DATA_BLOCK "RSE_DB"
TITLE = Report System Error Diagnostic Block
{ S7_Optimized_Access := 'FALSE' }
AUTHOR : SIMATIC
FAMILY : RSEDIAG
NAME : RSE4
VERSION : 1.0
NON_RETAIN
// This DB contains the generated data from STEP 7 Report System Errors.
"RSE_FB"

BEGIN
   w127Timer_a := BYTE#16#80;
   bAnwenderIO_Flag := BYTE#16#54;
   wRackEntry1 := WORD#16#0368;
   xFrei := TRUE;
   VFTable0_Hiera := BYTE#16#01;
   VFTable0_AsyncFct := BYTE#16#07;
   VFTable0_AsyncDat := BYTE#16#0F;
   VFTable0_SyncFct := BYTE#16#07;
   VFTable0_SyncDat := BYTE#16#0F;
   VFTable0_GehendDat := BYTE#16#0F;
   VFTable1_Hiera := BYTE#16#12;
   VFTable1_AsyncFct := BYTE#16#06;
   VFTable1_AsyncDat := BYTE#16#0D;
   VFTable1_SyncFct := BYTE#16#07;
   VFTable1_SyncDat := BYTE#16#0F;
   VFTable1_GehendDat := BYTE#16#0B;
   VFTable2_Peri := BYTE#16#10;
   VFTable2_Hiera := BYTE#16#12;
   VFTable2_AsyncDat := BYTE#16#01;
   VFTable2_SyncDat := BYTE#16#01;
   VFTable2_GehendDat := BYTE#16#0C;
   VFTable2_0C96Dat := BYTE#16#06;
   VFTable3_Hiera := BYTE#16#1A;
   VFTable3_AsyncFct := BYTE#16#07;
   VFTable3_AsyncDat := BYTE#16#0F;
   VFTable3_SyncFct := BYTE#16#07;
   VFTable3_SyncDat := BYTE#16#0F;
   VFTable3_GehendDat := BYTE#16#0F;
   VFTable3_0C96Dat := BYTE#16#0F;
   VFTable4_Hiera := BYTE#16#1B;
   VFTable4_AsyncFct := BYTE#16#07;
   VFTable4_AsyncDat := BYTE#16#0F;
   VFTable4_SyncFct := BYTE#16#07;
   VFTable4_SyncDat := BYTE#16#0F;
   VFTable4_GehendDat := BYTE#16#0F;
   VFTable4_0C96Dat := BYTE#16#0F;
   VFTable5_Peri := BYTE#16#10;
   VFTable5_Hiera := BYTE#16#12;
   VFTable5_AsyncDat := BYTE#16#01;
   VFTable5_SyncDat := BYTE#16#01;
   VFTable5_GehendDat := BYTE#16#0C;
   VFTable5_TextListIndex := BYTE#16#03;
   VFTable5_0C96Dat := BYTE#16#06;
   VFTable6_Peri := BYTE#16#02;
   VFTable6_Hiera := BYTE#16#12;
   VFTable6_AsyncFct := BYTE#16#04;
   VFTable6_AsyncDat := BYTE#16#09;
   VFTable6_SyncFct := BYTE#16#02;
   VFTable6_SyncDat := BYTE#16#08;
   VFTable6_GehendDat := BYTE#16#0C;
   VFTable6_TextListIndex := BYTE#16#03;
   VFTable7_Peri := BYTE#16#11;
   VFTable7_Hiera := BYTE#16#01;
   VFTable7_AsyncFct := BYTE#16#01;
   VFTable7_AsyncDat := BYTE#16#0F;
   VFTable7_SyncFct := BYTE#16#01;
   VFTable7_SyncDat := BYTE#16#0F;
   VFTable7_GehendDat := BYTE#16#0B;
   VFTable7_0C96Dat := BYTE#16#07;
   VFTable8_Peri := BYTE#16#09;
   VFTable8_Hiera := BYTE#16#01;
   VFTable8_AsyncFct := BYTE#16#01;
   VFTable8_AsyncDat := BYTE#16#04;
   VFTable8_SyncFct := BYTE#16#01;
   VFTable8_SyncDat := BYTE#16#04;
   VFTable8_GehendDat := BYTE#16#0B;
   VFTable8_0C96Dat := BYTE#16#07;
   VFTable9_Peri := BYTE#16#01;
   VFTable9_Hiera := BYTE#16#32;
   VFTable9_AsyncFct := BYTE#16#07;
   VFTable9_AsyncDat := BYTE#16#0F;
   VFTable9_SyncFct := BYTE#16#07;
   VFTable9_SyncDat := BYTE#16#0F;
   VFTable9_GehendDat := BYTE#16#0F;
   VFTable9_0C96Dat := BYTE#16#0F;
   VFTable10_Peri := BYTE#16#11;
   VFTable10_Hiera := BYTE#16#12;
   VFTable10_AsyncFct := BYTE#16#03;
   VFTable10_AsyncDat := BYTE#16#01;
   VFTable10_SyncFct := BYTE#16#03;
   VFTable10_SyncDat := BYTE#16#02;
   VFTable10_GehendDat := BYTE#16#0C;
   VFTable11_Peri := BYTE#16#09;
   VFTable11_Hiera := BYTE#16#12;
   VFTable11_AsyncFct := BYTE#16#06;
   VFTable11_AsyncDat := BYTE#16#0C;
   VFTable11_SyncFct := BYTE#16#06;
   VFTable11_SyncDat := BYTE#16#0C;
   VFTable11_GehendDat := BYTE#16#0C;
   VFTable12_Peri := BYTE#16#01;
   VFTable12_Hiera := BYTE#16#04;
   VFTable12_AsyncFct := BYTE#16#06;
   VFTable12_AsyncDat := BYTE#16#0A;
   VFTable12_SyncFct := BYTE#16#06;
   VFTable12_SyncDat := BYTE#16#0A;
   VFTable12_GehendDat := BYTE#16#0B;
   VFTable13_Peri := BYTE#16#01;
   VFTable13_Hiera := BYTE#16#04;
   VFTable13_AsyncFct := BYTE#16#06;
   VFTable13_AsyncDat := BYTE#16#0E;
   VFTable13_SyncFct := BYTE#16#06;
   VFTable13_SyncDat := BYTE#16#0E;
   VFTable13_GehendDat := BYTE#16#0E;
   ADA[1] := BYTE#16#01;
   TextListe[0] := DWORD#16#0001_8001;
   TextListe[1] := DWORD#16#0004_8004;
   TextListe[2] := DWORD#16#0003_8003;
   TextListe[3] := DWORD#16#8006_8006;
   wMapItemLogAdr_Ein_1 := WORD#16#0004;
   wMapItemLogAdr_Ein_2 := WORD#16#0008;
   wMapItemLogAdr_Ein_3 := WORD#16#000A;
   wMapItemLogAdr_Ein_4 := WORD#16#000C;
   wMapItemLogAdr_Ein_5 := WORD#16#000E;
   wMapItemLogAdr_Ein_6 := WORD#16#0010;
   wMapItemLogAdr_Ein_7 := WORD#16#0100;
   wMapItemLogAdr_Ein_8 := WORD#16#0110;
   wMapItemLogAdr_Ein_9 := WORD#16#0120;
   wMapItemLogAdr_Ein_10 := WORD#16#0130;
   wMapItemLogAdr_Ein_11 := WORD#16#0140;
   wMapItemLogAdr_Ein_12 := WORD#16#0150;
   wMapItemLogAdr_Ein_13 := WORD#16#0160;
   wMapItemLogAdr_Ein_14 := WORD#16#0162;
   wMapItemLogAdr_Ein_15 := WORD#16#0164;
   wMapItemLogAdr_Ein_16 := WORD#16#0166;
   wMapItemLogAdr_Ein_17 := WORD#16#0168;
   wMapItemLogAdr_Ein_18 := WORD#16#01A0;
   wMapItemLogAdr_Ein_19 := WORD#16#07FA;
   wMapItemLogAdr_Ein_20 := WORD#16#07FB;
   wMapItemLogAdr_Ein_21 := WORD#16#07FC;
   wMapItemLogAdr_Ein_22 := WORD#16#07FD;
   wMapItemLogAdr_Ein_23 := WORD#16#07FE;
   wMapItemLogAdr_Ein_24 := WORD#16#07FF;
   wMapItemLogAdr_Aus_1 := WORD#16#0001;
   wMapItemLogAdr_Aus_2 := WORD#16#0003;
   wMapItemLogAdr_Aus_3 := WORD#16#0005;
   wMapItemLogAdr_Aus_4 := WORD#16#000C;
   wMapItemLogAdr_Aus_5 := WORD#16#000E;
   wMapItemLogAdr_KAd_0 := WORD#16#0190;
   wMapItemLogAdr_KAd_1 := WORD#16#CFFF;
   wMapItemLogAdr_KAd_2 := WORD#16#FFF6;
   wMapItemLogAdr_KAd_3 := WORD#16#FFF7;
   wMapItemLogAdr_KAd_4 := WORD#16#FFF8;
   wMapItemLogAdr_KAd_5 := WORD#16#FFF9;
   wMapItemLogAdr_KAd_6 := WORD#16#FFFA;
   wMapItemLogAdr_KAd_7 := WORD#16#FFFB;
   wMapItemLogAdr_KAd_8 := WORD#16#FFFC;
   wMapItemLogAdr_KAd_9 := WORD#16#FFFD;
   wMapItemOffset_Ein_0 := WORD#16#016A;
   wMapItemOffset_Ein_1 := WORD#16#017F;
   wMapItemOffset_Ein_2 := WORD#16#0213;
   wMapItemOffset_Ein_3 := WORD#16#025B;
   wMapItemOffset_Ein_4 := WORD#16#02A3;
   wMapItemOffset_Ein_5 := WORD#16#01CB;
   wMapItemOffset_Ein_6 := WORD#16#02EB;
   wMapItemOffset_Ein_7 := WORD#16#00A1;
   wMapItemOffset_Ein_8 := WORD#16#00B6;
   wMapItemOffset_Ein_9 := WORD#16#00CB;
   wMapItemOffset_Ein_10 := WORD#16#00E0;
   wMapItemOffset_Ein_11 := WORD#16#00F5;
   wMapItemOffset_Ein_12 := WORD#16#010A;
   wMapItemOffset_Ein_13 := WORD#16#0281;
   wMapItemOffset_Ein_14 := WORD#16#01A9;
   wMapItemOffset_Ein_15 := WORD#16#01F1;
   wMapItemOffset_Ein_16 := WORD#16#0239;
   wMapItemOffset_Ein_17 := WORD#16#02C9;
   wMapItemOffset_Ein_18 := WORD#16#0131;
   wMapItemOffset_Ein_19 := WORD#16#015A;
   wMapItemOffset_Ein_20 := WORD#16#0146;
   wMapItemOffset_Ein_21 := WORD#16#0089;
   wMapItemOffset_Ein_22 := WORD#16#0071;
   wMapItemOffset_Ein_23 := WORD#16#0058;
   wMapItemOffset_Ein_24 := WORD#16#0311;
   wMapItemOffset_Aus_0 := WORD#16#0194;
   wMapItemOffset_Aus_1 := WORD#16#0226;
   wMapItemOffset_Aus_2 := WORD#16#026E;
   wMapItemOffset_Aus_3 := WORD#16#02FE;
   wMapItemOffset_Aus_4 := WORD#16#02B6;
   wMapItemOffset_Aus_5 := WORD#16#01DE;
   wMapItemOffset_KAd_0 := WORD#16#011F;
   wMapItemOffset_KAd_1 := WORD#16#002C;
   wMapItemOffset_KAd_2 := WORD#16#02DB;
   wMapItemOffset_KAd_3 := WORD#16#032A;
   wMapItemOffset_KAd_4 := WORD#16#024B;
   wMapItemOffset_KAd_5 := WORD#16#0293;
   wMapItemOffset_KAd_6 := WORD#16#0203;
   wMapItemOffset_KAd_7 := WORD#16#01BB;
   wMapItemOffset_KAd_8 := WORD#16#0046;
   wMapItemOffset_KAd_9 := WORD#16#0010;
   bMapItemDB_Ein_0 := WORD#16#050A;
   bMapItemDB_Ein_1 := WORD#16#050A;
   bMapItemDB_Ein_2 := WORD#16#050B;
   bMapItemDB_Ein_3 := WORD#16#050B;
   bMapItemDB_Ein_4 := WORD#16#050B;
   bMapItemDB_Ein_5 := WORD#16#050B;
   bMapItemDB_Ein_6 := WORD#16#050B;
   bMapItemDB_Ein_7 := WORD#16#0102;
   bMapItemDB_Ein_8 := WORD#16#0102;
   bMapItemDB_Ein_9 := WORD#16#0102;
   bMapItemDB_Ein_10 := WORD#16#0102;
   bMapItemDB_Ein_11 := WORD#16#0102;
   bMapItemDB_Ein_12 := WORD#16#0102;
   bMapItemDB_Ein_13 := WORD#16#0408;
   bMapItemDB_Ein_14 := WORD#16#0408;
   bMapItemDB_Ein_15 := WORD#16#0408;
   bMapItemDB_Ein_16 := WORD#16#0408;
   bMapItemDB_Ein_17 := WORD#16#0408;
   bMapItemDB_Ein_18 := WORD#16#0102;
   bMapItemDB_Ein_19 := WORD#16#0509;
   bMapItemDB_Ein_20 := WORD#16#0407;
   bMapItemDB_Ein_21 := WORD#16#0206;
   bMapItemDB_Ein_22 := WORD#16#0206;
   bMapItemDB_Ein_23 := WORD#16#0205;
   bMapItemDB_Ein_24 := WORD#16#030C;
   bMapItemDB_Aus_0 := WORD#16#050A;
   bMapItemDB_Aus_1 := WORD#16#050B;
   bMapItemDB_Aus_2 := WORD#16#050B;
   bMapItemDB_Aus_3 := WORD#16#050B;
   bMapItemDB_Aus_4 := WORD#16#050B;
   bMapItemDB_Aus_5 := WORD#16#050B;
   bMapItemDB_KAd_0 := WORD#16#0103;
   bMapItemDB_KAd_1 := WORD#16#0101;
   bMapItemDB_KAd_2 := WORD#16#0509;
   bMapItemDB_KAd_3 := WORD#16#020D;
   bMapItemDB_KAd_4 := WORD#16#0509;
   bMapItemDB_KAd_5 := WORD#16#0509;
   bMapItemDB_KAd_6 := WORD#16#0509;
   bMapItemDB_KAd_7 := WORD#16#0509;
   bMapItemDB_KAd_8 := WORD#16#0204;
   wMapItemSubstAdr_0 := WORD#16#FFFF;
   wMapItemSubstAdr_1 := WORD#16#FFFF;
   wMapItemSubstAdr_2 := WORD#16#FFFF;
   wMapItemSubstAdr_3 := WORD#16#FFFF;
   wMapItemSubstAdr_4 := WORD#16#FFFF;
   wMapItemSubstAdr_5 := WORD#16#FFFF;
   wMapItemSubstAdr_6 := WORD#16#FFFF;
   wMapItemSubstAdr_7 := WORD#16#FFFF;
   wMapItemSubstAdr_8 := WORD#16#FFFF;
   wMapItemSubstAdr_9 := WORD#16#FFFF;
   bAnzahlFreieEintraege := BYTE#16#1F;
   MeldungBandBreite_01 := BYTE#16#0A;
   Meldung_02 := WORD#16#1B5C;
   MeldungBandBreite_02 := BYTE#16#0A;
   Meldung_03 := WORD#16#1BCC;
   MeldungBandBreite_03 := BYTE#16#0A;
   Meldung_04 := WORD#16#1B5E;
   MeldungBandBreite_04 := BYTE#16#0A;
   Meldung_05 := WORD#16#1B5B;
   MeldungBandBreite_05 := BYTE#16#2E;
   Meldung_06 := WORD#16#1C70;
   MeldungBandBreite_06 := BYTE#16#18;
   Meldung_07 := WORD#16#1C73;
   MeldungBandBreite_07 := BYTE#16#18;
   Meldung_08 := WORD#16#1C6D;
   MeldungBandBreite_08 := BYTE#16#10;
   Meldung_09 := WORD#16#1BCE;
   MeldungBandBreite_09 := BYTE#16#10;
   Meldung_10 := WORD#16#1B59;
   MeldungBandBreite_10 := BYTE#16#90;
   xSubOrdinateStateOld := WORD#16#FFFF;
   xASVeraltet := WORD#16#FFFF;
   bASZyklusZaehler := BYTE#16#03;
   xAnlaufMilde := TRUE;

END_DATA_BLOCK

